TYPE ST_BaseCommunicatorStack :
STRUCT
	stMessage					: ST_BaseCommunicatorMassege;
	bSent						: BOOL;		//wysłane
	bConfirmation				: BOOL;		//potwierdzenie
	itfSender					: ITF_BaseMessengerSender;
	itfRecipient				: ITF_BaseMessengerRecipient;
	
END_STRUCT
END_TYPE

(* stored: Version 1.1.0.1
   DUT ST_BaseCommunicatorStack: Id {f3df0a22-2d82-062c-18b5-7c2b5a82b67e} *)
